FUNCTION_BLOCK GantryStatus
VAR_INPUT
	En: BOOL;	
	Paus: BOOL;
END_VAR
VAR_OUTPUT
	Auto : BOOL;
	ManualMode : BOOL;	
	Status : STRING;
END_VAR
VAR_IN_OUT
	Data:CommunicationData;
END_VAR
VAR
	fbTonStartDelay: TON;
END_VAR


fbTonStartDelay( IN := Data.Auto, PT := T#1S);


Auto 		:= fbTonStartDelay.Q;
ManualMode 	:= Data.ManualMode;
Status 		:= Data.Status;
Data.Paus := Paus;

END_FUNCTION_BLOCK

(* stored: Version 1.1.0.1, ProductVersion 3.1.4022.12
   POU GantryStatus: Id {3aa1aa55-45ed-45b7-a62c-325b2077c7ca}, SpecialFunc None *)
